{attribute 'GeneratedUsingTerminal: EL3351-0000-0016'}
{attribute addProperty BoxType "EL3351-0000-0016"}
{attribute addProperty Id "EtcSlaveTerminalBaseAIBridge_InputsAT %I*AIBridge_Inputs_555AA1E89AISupply_InputsAT %I*AISupply_Inputs_555AA1E89WcStateAT %I*WcState_9091E0EB2InfoDataAT %I*InfoData_32EB74EA10"}
{attribute addProperty CRC "371360226"}
{attribute addProperty Size "30"}
TYPE EL3351_162281E2 EXTENDS EtcSlaveTerminalBase :
STRUCT
	{attribute addProperty Name "AIBridge_Inputs"}
	AIBridge_Inputs : AIBridge_Inputs_555AA1E8;
	{attribute addProperty Name "AISupply_Inputs"}
	AISupply_Inputs : AISupply_Inputs_555AA1E8;
	{attribute addProperty Name "WcState"}
	WcState : WcState_9091E0EB;
	{attribute addProperty Name "InfoData"}
	InfoData : InfoData_32EB74EA;
END_STRUCT
END_TYPE

(* stored: Version 1.2.0.0, ProductVersion 3.1.4024.9
   DUT EL3351_162281E2: Id {3532fbe1-e2c3-49e1-8322-abad0f62f4d2} *)
